// TIA Portal V16 export
// export: Created 2024-12-03T15:41:44.2954097Z, ExportSetting WithDefaults, DisplayName Totally Integrated Automation Portal, DisplayVersion V16 Update 6, DisplayName TIA Portal Version Control Interface, DisplayVersion V16 Update 2, DisplayName TIA Portal Openness, DisplayVersion V16 Update 6, DisplayName TIA Portal Teamcenter Gateway, DisplayVersion V16, DisplayName SINAMICS Startdrive Advanced, DisplayVersion V16 Update 5, DisplayName SINAMICS Startdrive G130, G150, S120, S150, SINAMICS MV, S210, DisplayVersion V16 Update 5, DisplayName SINAMICS Startdrive G110M, G120, G120C, G120D, G120P, G115D, DisplayVersion V16 Update 5, DisplayName STEP 7 Professional, DisplayVersion V16 Update 6, DisplayName STEP 7 Safety, DisplayVersion V16, DisplayName WinCC Advanced / Unified PC, DisplayVersion V16 Update 6
DATA_BLOCK "MOT_CLX_DB"   // DB103
{ S7_Optimized_Access := 'FALSE' }
VERSION : 0.1
// stored: AutoNumber true, DBAccessibleFromOPCUA true, IsOnlyStoredInLoadMemory false, IsWriteProtectedInAS false
   VAR
      MOT_102L : "ConveyLinx_FullPLC_Single";
      MOT_102R : "ConveyLinx_FullPLC_Single";
      MOT_103L : "ConveyLinx_FullPLC_Single";
      MOT_103R : "ConveyLinx_FullPLC_Single";
      MOT_104L : "ConveyLinx_FullPLC_Single";
      MOT_104R : "ConveyLinx_FullPLC_Single";
      MOT_105L : "ConveyLinx_FullPLC_Single";
      MOT_105R : "ConveyLinx_FullPLC_Single";
      MOT_106L : "ConveyLinx_FullPLC_Single";
      MOT_106R : "ConveyLinx_FullPLC_Single";
      MOT_107L : "FLOWSORT_TWISTER_UDT";
      MOT_107R : "ConveyLinx_FullPLC_Single";
      MOT_108L : "ConveyLinx_FullPLC_Single";
      MOT_108R : "ConveyLinx_FullPLC_Single";
      MOT_109L : "ConveyLinx_FullPLC_Single";
      MOT_109R : "ConveyLinx_FullPLC_Single";
      MOT_110L : "ConveyLinx_FullPLC_Single";
      MOT_110R : "ConveyLinx_FullPLC_Single";
      MOT_111L : "ConveyLinx_FullPLC_Single";
      MOT_111R : "ConveyLinx_FullPLC_Single";
      MOT_112L : "ConveyLinx_FullPLC_Single";
      MOT_112R : "ConveyLinx_FullPLC_Single";
      MOT_113L : "ConveyLinx_FullPLC_Single";
      MOT_113R : "ConveyLinx_FullPLC_Single";
      MOT_114L : "ConveyLinx_FullPLC_Single";
      MOT_114R : "ConveyLinx_FullPLC_Single";
      MOT_115L : "ConveyLinx_FullPLC_Single";
      MOT_115R : "ConveyLinx_FullPLC_Single";
      MOT_201R_Belts { S7_SetPoint := 'True'} : "ConveyLinx_FullPLC_Single";
      MOT_201L_Lift { S7_SetPoint := 'True'} : "EasySystems_LineairMotor_ConveyLinx_FullPLC_Single";
      MOT_202L : "ConveyLinx_FullPLC_Single";
      MOT_202R : "ConveyLinx_FullPLC_Single";
      MOT_203L_Lift : "EasySystems_LineairMotor_ConveyLinx_FullPLC_Single";
      MOT_203R_Belts : "ConveyLinx_FullPLC_Single";
      MOT_301L : "ConveyLinx_FullPLC_Single";
      MOT_301R : "ConveyLinx_FullPLC_Single";
      MOT_302L : "ConveyLinx_FullPLC_Single";
      MOT_302R : "ConveyLinx_FullPLC_Single";
      MOT_303L : "ConveyLinx_FullPLC_Single";
      MOT_303R : "ConveyLinx_FullPLC_Single";
      MOT_304L : "ConveyLinx_FullPLC_Single";
      MOT_304R : "ConveyLinx_FullPLC_Single";
      MOT_305L : "ConveyLinx_FullPLC_Single";
      MOT_305R : "ConveyLinx_FullPLC_Single";
   END_VAR
BEGIN
END_DATA_BLOCK
